// TIA Portal V16 export
// export: Created 2024-09-05T17:39:19.5396244Z, ExportSetting WithDefaults, DisplayName Totally Integrated Automation Portal, DisplayVersion V16 Update 6, DisplayName TIA Portal Version Control Interface, DisplayVersion V16 Update 2, DisplayName TIA Portal Openness, DisplayVersion V16 Update 6, DisplayName STEP 7 Professional, DisplayVersion V16 Update 6, DisplayName STEP 7 Safety, DisplayVersion V16, DisplayName WinCC Advanced, DisplayVersion V16 Update 6
DATA_BLOCK "HMIData"   // DB1
{ S7_Optimized_Access := 'TRUE' }
VERSION : 0.1
// stored: AutoNumber false, DBAccessibleFromOPCUA true, IsOnlyStoredInLoadMemory false, IsRetainMemResEnabled false, IsWriteProtectedInAS false, MemoryReserve 100
   VAR
      HMI { S7_SetPoint := 'True'} : "UDT_HMI";
      ManualCommandHMI : Int := 0;
      ManualCommand : Int := 0;
   END_VAR
BEGIN
   HMI.ScreenData[1..5] := 16#0000;
   HMI.UserNumber := 0;
   HMI.ActualScreenNumber := 0;
   HMI.RequiredScreenNumber := 0;
   HMI.FunctionKeys[1..8] := FALSE;
END_DATA_BLOCK
